# EPICS StreamDevice protocol: ioc/protocol/micro820.proto
OutTerminator = CR;
InTerminator  = CR;
ReplyTimeout  = 600;

test    { out "TEST";   in "%d"}
